FUNCTION_BLOCK TMS_Mover EXTENDS FB_Mover IMPLEMENTS ITmsMover
VAR
	ActivateATrack : ActivateTrackForMover(_Axis);
	mcReadTrackPositions : Tc3_McCollisionAvoidance.MC_ReadTrackPositions;
	axesMoveModuloTo 		: MoveModuloMoverToPosition(_Axis) := (Gap := 100.0);
	_stOptions : ST_MoveAbsoluteCAOptions;
	ipTcIoXtsMover			: I_TcIoXtsXpuMover;
	stTmsActPositions			: ST_PositionInfo;
END_VAR

{analysis -2}

METHOD ActivateTrack : BOOL
VAR_INPUT
	newTrack : OTCID;
END_VAR
IF NOT ActivateATrack.Busy THEN
	ActivateATrack.Execute(Track := newTrack);
	ActivateTrack := TRUE;
ELSE
	ActivateTrack := FALSE;
END_IF
END_METHOD

PROPERTY ActiveTrack : OTCID
GET
ActiveTrack := stTmsActPositions.nTrackObjectid;
END_GET
END_PROPERTY

METHOD PUBLIC  Cycle : HRESULT
VAR_INPUT
END_VAR
Cycle := SUPER^.Cycle();
IF _identInGroup <> 0 THEN
	mcReadTrackPositions(
		Axis:= THIS^._Axis, 
		Enable:= TRUE, 
		Valid=> , 
		Busy=> , 
		TrackPosition=> , 
		TrackId=> , 
		PartPosition=> , 
		PartId=> , 
		Error=> , 
		ErrorId=> );
END_IF
Cycle := ActivateATrack.Cycle();
IF ActivateATrack.Done THEN 
	_stOptions.PositionReferenceSystem :=  ActivateATrack.NewTrackId;
	axesMoveModuloTo.Options := _stOptions;
END_IF

IF ipTcIoXtsMover <> 0 THEN
	stTmsActPositions:=ipTcIoXtsMover.GetPositionInfo();
END_IF
//bob := 
//ipTcIoXtsMover.GetActiveTrackObjectId();

Cycle := axesMoveModuloTo.Cycle();
END_METHOD

METHOD PUBLIC HasCommand : BOOL
VAR_INPUT
END_VAR
HasCommand := axesMoveModuloTo.Busy;
END_METHOD

METHOD isAtPosition : BOOL
VAR_INPUT
	position : MC_LREAL;
END_VAR
//Create modulo position 
IF position > 1 THEN
	IF stTmsActPositions.fTrackPosition < position + 1 AND stTmsActPositions.fTrackPosition > position - 1 THEN
		isAtPosition := TRUE;
	ELSE
		isAtPosition := FALSE;
	END_IF  
ELSE
	IF stTmsActPositions.fTrackPosition < position + 1 AND stTmsActPositions.fTrackPosition > 0.0  
		OR stTmsActPositions.fTrackPosition < _trackLength AND stTmsActPositions.fTrackPosition > _trackLength - 1 THEN
		isAtPosition := TRUE;
	ELSE
		isAtPosition := FALSE;
	END_IF
END_IF
END_METHOD

METHOD PUBLIC isPastPosition : BOOL
VAR_INPUT
	position : MC_LREAL;
END_VAR
IF position > 1 THEN
	IF stTmsActPositions.fTrackPosition > position THEN
		isPastPosition := TRUE;
	ELSE
		isPastPosition := FALSE;
	END_IF  
ELSE
	isPastPosition := FALSE;
END_IF
END_METHOD

METHOD PUBLIC MoveTo : BOOL
VAR_INPUT
	Position : MC_LREAL;
	Velocity : MC_LREAL;
	BackwardMove : BOOL; //NOT USED IN THIS CALL
END_VAR
IF NOT THIS^.isAtPosition(position := Position) THEN
	IF NOT axesMoveModuloTo.Busy THEN
		THIS^.axesMoveModuloTo.MoveTo(Position := Position, Velocity := Velocity, Direction := Tc2_MC2.MC_Direction.MC_Positive_Direction, Turns := 0);
		MoveTo := TRUE;
		_targetPos := Position;
	ELSE
		MoveTo := FALSE;
	END_IF
ELSE
	MoveTo := FALSE;
END_IF
END_METHOD

METHOD PUBLIC SetMoverInterface : BOOL
VAR_INPUT
	MoverInterface : I_TcIoXtsXpuMover;
END_VAR
ipTcIoXtsMover := MoverInterface;
SetMoverInterface := TRUE;
END_METHOD

END_FUNCTION_BLOCK

(* stored: Version 1.1.0.1, ProductVersion 3.1.4024.12
   POU TMS_Mover: Id {5460a3ca-ef4a-4eb7-aee0-351ddb8da841}, SpecialFunc None
   Method ActivateTrack: Id {67dea5a7-1ddb-45ab-b6fb-8140fc4e28a1}
   Property ActiveTrack: Id {8713b95c-1a45-4154-9f81-8eda6eb00e1d}
   Get Get: Id {b47e9603-d05b-4fb2-8c08-570f9ee8994f}
   Method Cycle: Id {1d05da50-72aa-4e35-9556-57a03180f6ab}
   Method HasCommand: Id {ed907035-91a3-47dc-9314-24c9235dbc23}
   Method isAtPosition: Id {1ca12edb-5e3c-438e-86ce-3f842724e28c}
   Method isPastPosition: Id {40eb8c66-39fe-4229-9666-f2ee6f651513}
   Method MoveTo: Id {0eb6ed83-3f5e-4a80-9c66-5b86c77ea5cc}
   Method SetMoverInterface: Id {e0a200ba-97fb-445b-94c1-a82a08618f42} *)
